
// ===== library types =====

// folder: Modbus Polling Engine

TYPE "typeMasterData"
VERSION : 0.1
   STRUCT
      Done : Bool;
      Busy : Bool;
      Error : Bool;
      locked : Bool;
      Mode : USInt;
      Status : Int;
      "Slave ID" : UInt;
      "Register Address" : UDInt;
      Length : UInt;
      RequestID : UInt;
      Data : Array[0..299] of Byte;
   END_STRUCT;
END_TYPE

// folder: (top level)

FUNCTION_BLOCK "PollTosibox"   // FB1, SCL
{ S7_Optimized_Access := 'TRUE' }
VERSION : 0.1
   VAR_INPUT
      slaveId : Int;   // modbus slave id
   END_VAR
   VAR_OUTPUT
      latitude : LReal;
      longitude : LReal;
      UTCTime : LReal;
   END_VAR
   VAR_IN_OUT
      modbusInterface : "typeMasterData";
   END_VAR
   VAR
      statData : Array[0..11] of Int;
      statLat : Array[0..7] of Byte;
      statLon : Array[0..7] of Byte;
      statUTC : Array[0..7] of Byte;
   END_VAR
   VAR_TEMP
      tempStatus : Int;
      tempPos : DInt;
   END_VAR
BEGIN
   //=============================================================================
   // AWC Inc.
   // (c)Copyright 2015 All Rights Reserved
   //-----------------------------------------------------------------------------
   // Library: (that the source is dedicated to)
   // Tested with: 1500 Family, 1200 Family
   // Engineering: TIA Portal v13 SP1 upd7
   // Restrictions: None
   // Requirements: s7 1200 or 1500 family depending on number used
   // Functionality: Get Modbus Values from TosiMox
   // 
   // 
   // 
   // 
   //-----------------------------------------------------------------------------
   // Change log table:
   // 01.00.00 07/30/2020 Created by Matt Paulissen
   //=============================================================================
   //
   "LargeModbusPoll"(slaveId:=1,
                     address:=40001,
                     data=>#statData,
                     status=>#tempStatus,
                     modbusInterface:=#modbusInterface);
   //Parse Latitude
   #statLat[0] := #statData[3].%B1;
   #statLat[1] := #statData[3].%B0;
   #statLat[2] := #statData[2].%B1;
   #statLat[3] := #statData[2].%B0;
   #statLat[4] := #statData[1].%B1;
   #statLat[5] := #statData[1].%B0;
   #statLat[6] := #statData[0].%B1;
   #statLat[7] := #statData[0].%B0;

   #tempPos := 0;
   #tempStatus := Deserialize(SRC_ARRAY := #statLat, DEST_VARIABLE => #latitude, POS := #tempPos);
   //Parse Longitude
   #statLon[0] := #statData[7].%B1;
   #statLon[1] := #statData[7].%B0;
   #statLon[2] := #statData[6].%B1;
   #statLon[3] := #statData[6].%B0;
   #statLon[4] := #statData[5].%B1;
   #statLon[5] := #statData[5].%B0;
   #statLon[6] := #statData[4].%B1;
   #statLon[7] := #statData[4].%B0;

   #tempPos := 0;
   #tempStatus := Deserialize(SRC_ARRAY := #statLon, DEST_VARIABLE => #longitude, POS := #tempPos);

   //Parse Time
   #statUTC[0] := #statData[11].%B1;
   #statUTC[1] := #statData[11].%B0;
   #statUTC[2] := #statData[10].%B1;
   #statUTC[3] := #statData[10].%B0;
   #statUTC[4] := #statData[9].%B1;
   #statUTC[5] := #statData[9].%B0;
   #statUTC[6] := #statData[8].%B1;
   #statUTC[7] := #statData[8].%B0;

   #tempPos := 0;
   #tempStatus := Deserialize(SRC_ARRAY := #statUTC, DEST_VARIABLE => #UTCTime, POS := #tempPos);
END_FUNCTION_BLOCK

FUNCTION "LargeModbusPoll" : Void   // FC892, SCL
{ S7_Optimized_Access := 'TRUE' }
VERSION : 0.1
   VAR_INPUT
      slaveId : Int;   // modbus slave id
      address : UInt;   // starting modbus register address
   END_VAR
   VAR_OUTPUT
      data : Variant;   // <uint><int><word><dword><real>
      status : Int;   // status of modbus read
   END_VAR
   VAR_IN_OUT
      modbusInterface : "typeMasterData";
   END_VAR
   VAR_TEMP
      tempPosition : DInt;
      tempStatus : Int;
      tempMode : USInt;
      tempAddress : UInt;
   END_VAR
BEGIN
   //=============================================================================
   // AWC Inc.
   // (c)Copyright 2018 All Rights Reserved
   //-----------------------------------------------------------------------------
   // Library: (that the source is dedicated to)
   // Tested with: 1500 Family, 1200 Family
   // Engineering: TIA Portal v13 SP1 upd7
   // Restrictions: None
   // Requirements: s7 1200 or 1500 family depending on number used
   // Functionality: Get Modbus Input Variant UDT
   // 
   // 
   // 
   // 
   //-----------------------------------------------------------------------------
   // Change log table:
   // 01.00.00 05/17/2018 Created by Matt Paulissen
   // 01.00.02 09/21/2018 Added request ID to detect stuck lock
   // 01.01.06 09/29/2020 Added extended modbus addressing
   //=============================================================================

   //Check for lock
   IF (NOT #modbusInterface.locked) THEN
       //Move Register and Slave address to Modbus Register
       #modbusInterface."Slave ID" := #slaveId;
       #modbusInterface."Register Address" := #address;

       //Get UDT length in bytes
       #tempStatus := Serialize(SRC_VARIABLE := #data, DEST_ARRAY => #modbusInterface.Data, POS := #tempPosition);
       IF (#tempStatus <> 0) THEN  //Exit instruction if UDT cannot be processed by the modbus interface
           RETURN;
       END_IF;
       //Get number of registers needed to poll entire UDT
       CASE #address OF
           1..9999, 10001..19999:  //Edge case for boolean values
               #tempPosition := #tempPosition * 8; //Multiply bytes by 8 to get bits
           50000..59999:  //Edge case for extended addressing
               #modbusInterface.Mode := 104;
               #modbusInterface."Register Address" := #address - 40001;
               IF ((#tempPosition MOD 2) = 0) THEN
                   #tempPosition := #tempPosition / 2;
               ELSE
                   #tempPosition := (#tempPosition / 2) + 1;
               END_IF;
           ELSE  //Normal registers
               #modbusInterface.Mode := 0;
               IF ((#tempPosition MOD 2) = 0) THEN
                   #tempPosition := #tempPosition / 2;
               ELSE
                   #tempPosition := (#tempPosition / 2) + 1;
               END_IF;
       END_CASE;
       #modbusInterface.Length := #tempPosition;
       #modbusInterface.locked := TRUE;
       #modbusInterface.RequestID += 1;
       RETURN;
   END_IF;
   //Edge case handling for extended modbus addressing
   IF (#address >= 50000 AND #address <= 59999) THEN
       #tempAddress := #address - 40001;
       #tempMode := 104;
   ELSE
       #tempAddress := #address;
       #tempMode := 0;
   END_IF;
   IF ((#modbusInterface.locked)
       AND (
       (#modbusInterface."Slave ID" = #slaveId)
       AND (#modbusInterface."Register Address" = #tempAddress)
       AND (#modbusInterface.Mode = #tempMode))
       )
   THEN
       IF (#modbusInterface.Done) THEN
           //Deserialize to output
           #tempStatus := Deserialize(SRC_ARRAY := #modbusInterface.Data, DEST_VARIABLE => #data, POS := #tempPosition);
           #modbusInterface.locked := FALSE;
           #status := #modbusInterface.Status;
       END_IF;
       IF (#modbusInterface.Error) THEN
           //TODO: error handling for variant????
           #modbusInterface.locked := 0;
           #status := #modbusInterface.Status;
       END_IF;
   END_IF;
END_FUNCTION

FUNCTION "GeneralModbusWrite" : Void   // FC893, SCL
{ S7_Optimized_Access := 'TRUE' }
VERSION : 0.1
   VAR_INPUT
      slaveId : Int;   // modbus slave id
      address : UInt;   // starting modbus register address
      write : Bool;   // write data to register
      data : Variant;   // value to write to modbus register
      swappedFloatingPoint : Bool;   // set to true for word swapped floating point
   END_VAR
   VAR_OUTPUT
      status : Word;
   END_VAR
   VAR_IN_OUT
      modbusInterface : "typeMasterData";
   END_VAR
   VAR_TEMP
      tempdWord : DWord;
      tempUint : UInt;
      tempInt : Int;
      tempWord : Word;
      tempReal : Real;
      tempBool : Bool;
      tempStatus : Int;
      tempPos : DInt;
   END_VAR
   VAR CONSTANT
      WRITE_OK : Word := 16#7000;
   END_VAR
BEGIN
   //=============================================================================
   // AWC Inc.
   // (c)Copyright 2015 All Rights Reserved
   //-----------------------------------------------------------------------------
   // Library: (that the source is dedicated to)
   // Tested with: 1500 Family, 1200 Family
   // Engineering: TIA Portal v13 SP1 upd7
   // Restrictions: None
   // Requirements: s7 1200 or 1500 family depending on number used
   // Functionality: Get Modbus Input
   // 
   // 
   // 
   // 
   //-----------------------------------------------------------------------------
   // Change log table:
   // 01.00.00 08/09/2017 Created by Matt Paulissen
   // 01.00.01 08/23/2017 Added ability to set failover value
   // 01.00.02 09/21/2018 Added request ID to detect stuck lock
   // 01.01.01 01/25/2019 Added ability to write to coils
   // 01.01.07 03/16/2021 Bug Fix for writing single coil
   //=============================================================================

   //Check for lock
   IF ((NOT #modbusInterface.locked) AND (#write)) THEN
       //Move Register and Slave address to Modbus Register
       #modbusInterface."Slave ID" := #slaveId;
       #modbusInterface."Register Address" := #address;
       #modbusInterface.Mode := 1;
       CASE TypeOf(#data) OF
           UInt:
               #modbusInterface.Length := 1;
               //VariantGet(SRC:=#data,
               //           DST=>#tempUint);
               #tempStatus := Serialize(SRC_VARIABLE := #data, DEST_ARRAY => #modbusInterface.Data, POS := #tempPos);

               //#modbusInterface.Data[0] := #tempUint;
           Int:
               #modbusInterface.Length := 1;
               // VariantGet(SRC := #data,
               //            DST => #tempInt);
               // #modbusInterface.Data[0] := INT_TO_UINT(IN:=#tempInt);
               #tempStatus := Serialize(SRC_VARIABLE := #data, DEST_ARRAY => #modbusInterface.Data, POS := #tempPos);
           Word:
               #modbusInterface.Length := 1;
               // VariantGet(SRC := #data,
               //            DST => #tempWord);
               // #modbusInterface.Data[0] := WORD_TO_UINT(IN := #tempWord);
               #tempStatus := Serialize(SRC_VARIABLE := #data, DEST_ARRAY => #modbusInterface.Data, POS := #tempPos);
           DWord:
               #modbusInterface.Length := 2;
               VariantGet(SRC := #data,
                          DST => #tempdWord);
               IF #swappedFloatingPoint THEN
                   // Swapped 
                   #modbusInterface.Data[2] := #tempdWord.%B3;
                   #modbusInterface.Data[3] := #tempdWord.%B2;
                   #modbusInterface.Data[0] := #tempdWord.%B1;
                   #modbusInterface.Data[1] := #tempdWord.%B0;
               ELSE
                   //Consecutive
                   #modbusInterface.Data[3] := #tempdWord.%B0;
                   #modbusInterface.Data[2] := #tempdWord.%B1;
                   #modbusInterface.Data[1] := #tempdWord.%B2;
                   #modbusInterface.Data[0] := #tempdWord.%B3;
               END_IF;
           Real:
               #modbusInterface.Length := 2;
               VariantGet(SRC := #data,
                          DST => #tempReal);
               #tempdWord := REAL_TO_DWORD(IN:=#tempReal);
               IF #swappedFloatingPoint THEN
                   // Swapped 
                   #modbusInterface.Data[2] := #tempdWord.%B3;
                   #modbusInterface.Data[3] := #tempdWord.%B2;
                   #modbusInterface.Data[0] := #tempdWord.%B1;
                   #modbusInterface.Data[1] := #tempdWord.%B0;
               ELSE
                   //Consecutive
                   #modbusInterface.Data[3] := #tempdWord.%B0;
                   #modbusInterface.Data[2] := #tempdWord.%B1;
                   #modbusInterface.Data[1] := #tempdWord.%B2;
                   #modbusInterface.Data[0] := #tempdWord.%B3;
               END_IF;
           Bool:
               #modbusInterface.Length := 1;
               VariantGet(SRC := #data,
                          DST => #tempBool);
               // Cleared buffer to fix bug during single coil writes
               #modbusInterface.Data[0] := 0;
               #modbusInterface.Data[1] := 0;
               #modbusInterface.Data[0].%X0 := #tempBool;
           ELSE  // Statement section ELSE
               ;
       END_CASE;
       #modbusInterface.locked := TRUE;
       #modbusInterface.RequestID += 1;
       RETURN;
   END_IF;
   IF ((#modbusInterface.locked)
       AND (
       (#modbusInterface."Slave ID" = #slaveId)
       AND (#modbusInterface."Register Address" = #address)
       AND (#modbusInterface.Mode = 1))
       )
   THEN
       IF (#modbusInterface.Done) THEN
           //Inspect type of output and set correct type of input in modbus register
           #status := #WRITE_OK;
           #modbusInterface.locked := FALSE;
       END_IF;
       IF (#modbusInterface.Error) THEN
           #status := #modbusInterface.Status;
           #modbusInterface.locked := false;
       END_IF;
   END_IF;
END_FUNCTION

FUNCTION "Mag6/8000" : Void   // FC896, SCL
{ S7_Optimized_Access := 'TRUE' }
VERSION : 0.1
   VAR_INPUT
      slaveId : Int;   // modbus slave id
   END_VAR
   VAR_OUTPUT
      velocity : Variant;   // current velocity <real>
      flow : Variant;   // current flow <real>
      totalizer : Variant;   // totalizer <array[0..2] of UDINT>
   END_VAR
   VAR_IN_OUT
      modbusInterface : "typeMasterData";
   END_VAR
   VAR_TEMP
      tempStatus : Int;
   END_VAR
BEGIN
   //=============================================================================
   // AWC Inc.
   // (c)Copyright 2015 All Rights Reserved
   //-----------------------------------------------------------------------------
   // Library: (that the source is dedicated to)
   // Tested with: 1500 Family, 1200 Family
   // Engineering: TIA Portal v13 SP1 upd7
   // Restrictions: None
   // Requirements: s7 1200 or 1500 family depending on number used
   // Functionality: Get Modbus Values from Siemens Mag6000 or 8000
   // 
   // 
   // 
   // 
   //-----------------------------------------------------------------------------
   // Change log table:
   // 01.00.00 01/14/2019 Created by Matt Paulissen
   //=============================================================================
   //Current Velocity
   "GeneralModbusPoll"(slaveId:=#slaveId,
                       address:=42999,
                       swappedFloatingPoint:=false,
                       substituteValue:=0.0,
                       data=>#velocity,
                       modbusInterface:=#modbusInterface);
   //Current Flow
   "GeneralModbusPoll"(slaveId := #slaveId,
                       address := 43001,
                       swappedFloatingPoint := false,
                       substituteValue := 0.0,
                       data => #flow,
                       modbusInterface := #modbusInterface);
   //Totalizer
   "LargeModbusPoll"(slaveId:=#slaveId,
                     address:=43016
                     ,
                     data=>#totalizer,
                     status=> #tempStatus,
                     modbusInterface:=#modbusInterface);
END_FUNCTION

// folder: Cameron

FUNCTION "NuFlo" : Void   // FC897, SCL
{ S7_Optimized_Access := 'TRUE' }
VERSION : 0.1
   VAR_INPUT
      slaveId : Int;   // modbus slave id
   END_VAR
   VAR_OUTPUT
      currentFlow : Variant;   // current flow <real>
      currentTotal : Variant;   // current total <real>
      grandTotal : Variant;   // grand total <real>
   END_VAR
   VAR_IN_OUT
      modbusInterface : "typeMasterData";
   END_VAR
BEGIN
   //=============================================================================
   // AWC Inc.
   // (c)Copyright 2015 All Rights Reserved
   //-----------------------------------------------------------------------------
   // Library: (that the source is dedicated to)
   // Tested with: 1500 Family, 1200 Family
   // Engineering: TIA Portal v13 SP1 upd7
   // Restrictions: None
   // Requirements: s7 1200 or 1500 family depending on number used
   // Functionality: Get Modbus Values from Cameron Nu Flo
   // 
   // 
   // 
   // 
   //-----------------------------------------------------------------------------
   // Change log table:
   // 01.00.00 01/08/2019 Created by Matt Paulissen
   //=============================================================================
   //Current Flow
   "GeneralModbusPoll"(slaveId:=#slaveId,
                       address:=48013,
                       swappedFloatingPoint:=false,
                       substituteValue:=0.0,
                       data=>#currentFlow,
                       modbusInterface:=#modbusInterface);
   //Current Total
   "GeneralModbusPoll"(slaveId := #slaveId,
                       address := 48027,
                       swappedFloatingPoint := false,
                       substituteValue := 0.0,
                       data => #currentTotal,
                       modbusInterface := #modbusInterface);
   //Grand Total
   "GeneralModbusPoll"(slaveId := #slaveId,
                       address := 48011,
                       swappedFloatingPoint := false,
                       substituteValue := 0.0,
                       data => #grandTotal,
                       modbusInterface := #modbusInterface);
END_FUNCTION

// folder: ElectroLab

FUNCTION "LevelStick2100" : Void   // FC898, SCL
{ S7_Optimized_Access := 'TRUE' }
VERSION : 0.1
   VAR_INPUT
      slaveId : Int;   // modbus slave id
   END_VAR
   VAR_OUTPUT
      level : Variant;   // current level <uint>
      interfaceLevel : Variant;   // current interface level <uint>
   END_VAR
   VAR_IN_OUT
      modbusInterface : "typeMasterData";
   END_VAR
BEGIN
   //=============================================================================
   // AWC Inc.
   // (c)Copyright 2015 All Rights Reserved
   //-----------------------------------------------------------------------------
   // Library: (that the source is dedicated to)
   // Tested with: 1500 Family, 1200 Family
   // Engineering: TIA Portal v13 SP1 upd7
   // Restrictions: None
   // Requirements: s7 1200 or 1500 family depending on number used
   // Functionality: Get Modbus Values from Electrolab 2100
   // 
   // 
   // 
   // 
   //-----------------------------------------------------------------------------
   // Change log table:
   // 01.00.00 01/14/2019 Created by Matt Paulissen
   //=============================================================================
   //Current Velocity
   "GeneralModbusPoll"(slaveId:=#slaveId,
                       address:=43991,
                       swappedFloatingPoint:=false,
                       substituteValue:=0.0,
                       data=>#level,
                       modbusInterface:=#modbusInterface);
   "GeneralModbusPoll"(slaveId := #slaveId,
                       address := 43992,
                       swappedFloatingPoint := false,
                       substituteValue := 0.0,
                       data => #interfaceLevel,
                       modbusInterface := #modbusInterface);
END_FUNCTION

// folder: Modbus Polling Engine

FUNCTION_BLOCK "ModbusRtuEngine"   // FB6, LAD
{ S7_Optimized_Access := 'TRUE' }
VERSION : 0.1
// S7 1200 version of modbus polling engine.  Changed the Modbus Master to an MB_Master
   VAR_INPUT
      port : Port;
      baudRate : UDInt;
      parity : UInt;
      FirstScan : Bool;
      Reset : Bool;
   END_VAR
   VAR_OUTPUT
      Status : Int;
   END_VAR
   VAR_IN_OUT
      masterInterface : "typeMasterData";
   END_VAR
   VAR
      statPrevious : Int;
      statCurrent : Int;
      statIndex : Int;
      statRequestID : UInt;
      Comm_Load_Status : Int;
      Comm_Load_Done : Bool;
      Comm_Load_Error : Bool;
      instStuckInterfaceTimer : TON_TIME;
      instReinitilizeTimer : TON_TIME;
      instCommLoad : Modbus_Comm_Load;
      instMaster : Modbus_Master;
      inst7002Timeout : TON_TIME;
   END_VAR
   VAR_TEMP
      tempServerStatus : Int;
   END_VAR
   VAR CONSTANT
      UNITIALIZED : Int := 0;
      INITIALIZING_PORT : Int := 1;
      POLLING : Int := 2;
      POLLING_DONE : Int := 3;
   END_VAR
   VAR_TEMP   // added for the SCL form of the ladder/FBD networks
      _w1 : Bool;
   END_VAR
BEGIN

REGION Network 1: Run Comm Load
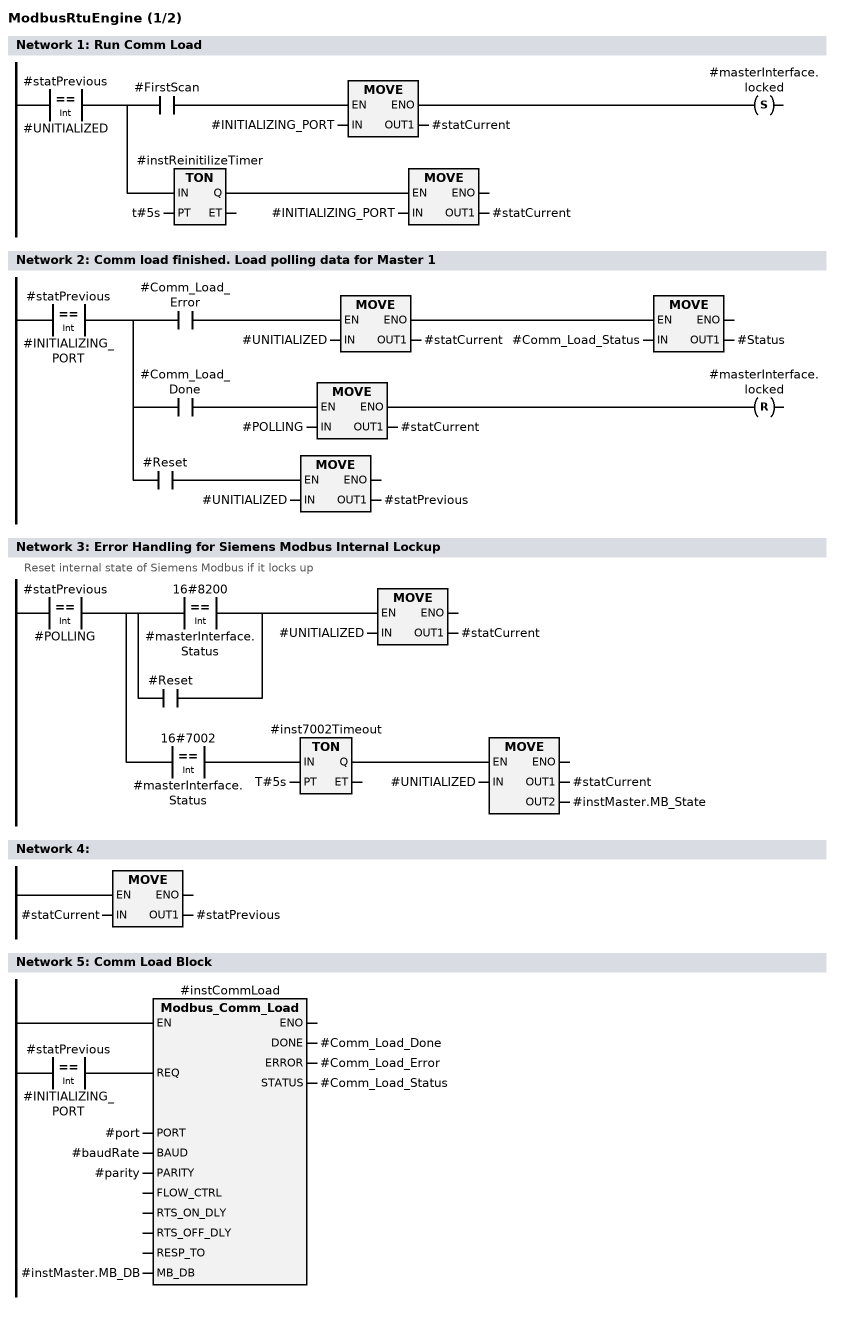
   #_w1 := #statPrevious = #UNITIALIZED;
   IF #_w1 AND #FirstScan THEN
       #statCurrent := #INITIALIZING_PORT;
       #masterInterface.locked := TRUE;
   END_IF;
   #instReinitilizeTimer(IN := #_w1, PT := t#5s);   // TON
   IF #instReinitilizeTimer.Q THEN #statCurrent := #INITIALIZING_PORT; END_IF;
END_REGION

REGION Network 2: Comm load finished. Load polling data for Master 1
   RUNG wire#powerrail
      { S7_Templates := "SrcType := Int" } EQ_Contact(in1 := #statPrevious, in2 := #INITIALIZING_PORT)
      wire#w1
      Contact( #Comm_Load_Error )
      Move(in := #UNITIALIZED, out1 => #statCurrent)
      Move(in := #Comm_Load_Status, out1 => #Status)
   END_RUNG
   RUNG wire#w1
      Contact( #Comm_Load_Done )
      Move(in := #POLLING, out1 => #statCurrent)
      R_Coil( #masterInterface.locked )
   END_RUNG
   RUNG wire#w1
      Contact( #Reset )
      Move(in := #UNITIALIZED, out1 => #statPrevious)
   END_RUNG
   // the same network as SCL:
   #_w1 := #statPrevious = #INITIALIZING_PORT;
   IF #_w1 AND #Comm_Load_Error THEN
       #statCurrent := #UNITIALIZED;
       #Status := #Comm_Load_Status;
   END_IF;
   IF #_w1 AND #Comm_Load_Done THEN
       #statCurrent := #POLLING;
       #masterInterface.locked := FALSE;
   END_IF;
   IF #_w1 AND #Reset THEN #statPrevious := #UNITIALIZED; END_IF;
END_REGION

REGION Network 3: Error Handling for Siemens Modbus Internal Lockup
   // Reset internal state of Siemens Modbus if it locks up
   #_w1 := #statPrevious = #POLLING;
   IF #_w1 AND ((16#8200 = #masterInterface.Status) OR #Reset) THEN #statCurrent := #UNITIALIZED; END_IF;
   #inst7002Timeout(IN := #_w1 AND (16#7002 = #masterInterface.Status), PT := T#5s);   // TON
   IF #inst7002Timeout.Q THEN
       #statCurrent := #UNITIALIZED;
       #instMaster.MB_State := #UNITIALIZED;
   END_IF;
END_REGION

REGION Network 4
   RUNG wire#powerrail
      Move(in := #statCurrent, out1 => #statPrevious)
   END_RUNG
   // the same network as SCL:
   #statPrevious := #statCurrent;
END_REGION

REGION Network 5: Comm Load Block
   #instCommLoad(REQ := #statPrevious = #INITIALIZING_PORT,   // Modbus_Comm_Load
                 PORT := #port,
                 BAUD := #baudRate,
                 PARITY := #parity,
                 MB_DB := #instMaster.MB_DB,
                 DONE => #Comm_Load_Done,
                 ERROR => #Comm_Load_Error,
                 STATUS => #Comm_Load_Status);
END_REGION

REGION Network 6: Master Instance 1
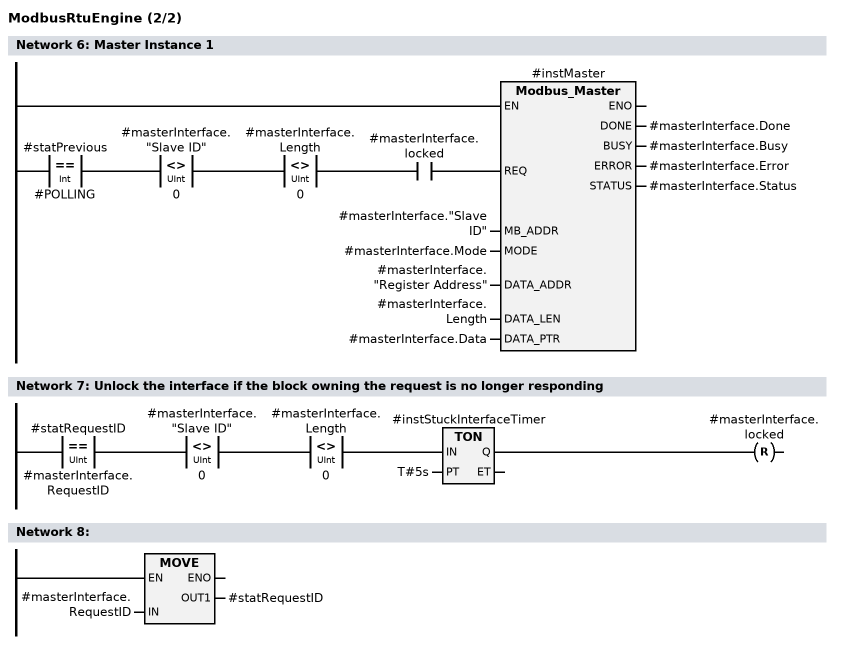
   #instMaster(REQ := (#statPrevious = #POLLING) AND (#masterInterface."Slave ID" <> 0) AND (#masterInterface.Length <> 0) AND #masterInterface.locked,   // Modbus_Master
               MB_ADDR := #masterInterface."Slave ID",
               MODE := #masterInterface.Mode,
               DATA_ADDR := #masterInterface."Register Address",
               DATA_LEN := #masterInterface.Length,
               DATA_PTR := #masterInterface.Data,
               DONE => #masterInterface.Done,
               BUSY => #masterInterface.Busy,
               ERROR => #masterInterface.Error,
               STATUS => #masterInterface.Status);
END_REGION

REGION Network 7: Unlock the interface if the block owning the request is no longer responding
   #instStuckInterfaceTimer(IN := (#statRequestID = #masterInterface.RequestID) AND (#masterInterface."Slave ID" <> 0) AND (#masterInterface.Length <> 0),   // TON
                           PT := T#5s);
   IF #instStuckInterfaceTimer.Q THEN #masterInterface.locked := FALSE; END_IF;
END_REGION

REGION Network 8
   RUNG wire#powerrail
      Move(in := #masterInterface.RequestID, out1 => #statRequestID)
   END_RUNG
   // the same network as SCL:
   #statRequestID := #masterInterface.RequestID;
END_REGION
END_FUNCTION_BLOCK

FUNCTION_BLOCK "ModbusTCPEngine"   // FB22, LAD
{ S7_Optimized_Access := 'TRUE' }
VERSION : 0.1
   VAR_INPUT
      port : Hw_Any;   // hardware identifier of port
      connectionId : Conn_Ouc;
      tcpPort : UInt;
      ipOne : Byte;   // ip octet one
      ipTwo : Byte;   // ip octet two
      ipThree : Byte;   // ip octet three
      ipFour : Byte;   // ip octet four
   END_VAR
   VAR_OUTPUT
      Status : Int;
   END_VAR
   VAR_IN_OUT
      masterInterface : "typeMasterData";
   END_VAR
   VAR
      instClient : MB_CLIENT;
      connection : TCON_IP_v4;
      statRequestID : UInt;
      instStuckInterfaceTimer : TON_TIME;
   END_VAR
   VAR CONSTANT
      UNITIALIZED : Int := 0;
      INITIALIZING_PORT : Int := 1;
      POLLING_ONE : Int := 2;
      POLLING_DONE_ONE : Int := 3;
      POLLING_TWO : Int := 4;
      POLLING_TWO_DONE : Int := 5;
   END_VAR
   // connection.ConnectionType := 11;
   // connection.ActiveEstablished := 1;
   // connection.RemotePort := 502;
   // connection.LocalPort := 502;
BEGIN

REGION Network 1: Move ip address from interface to static tcon_ip_v4
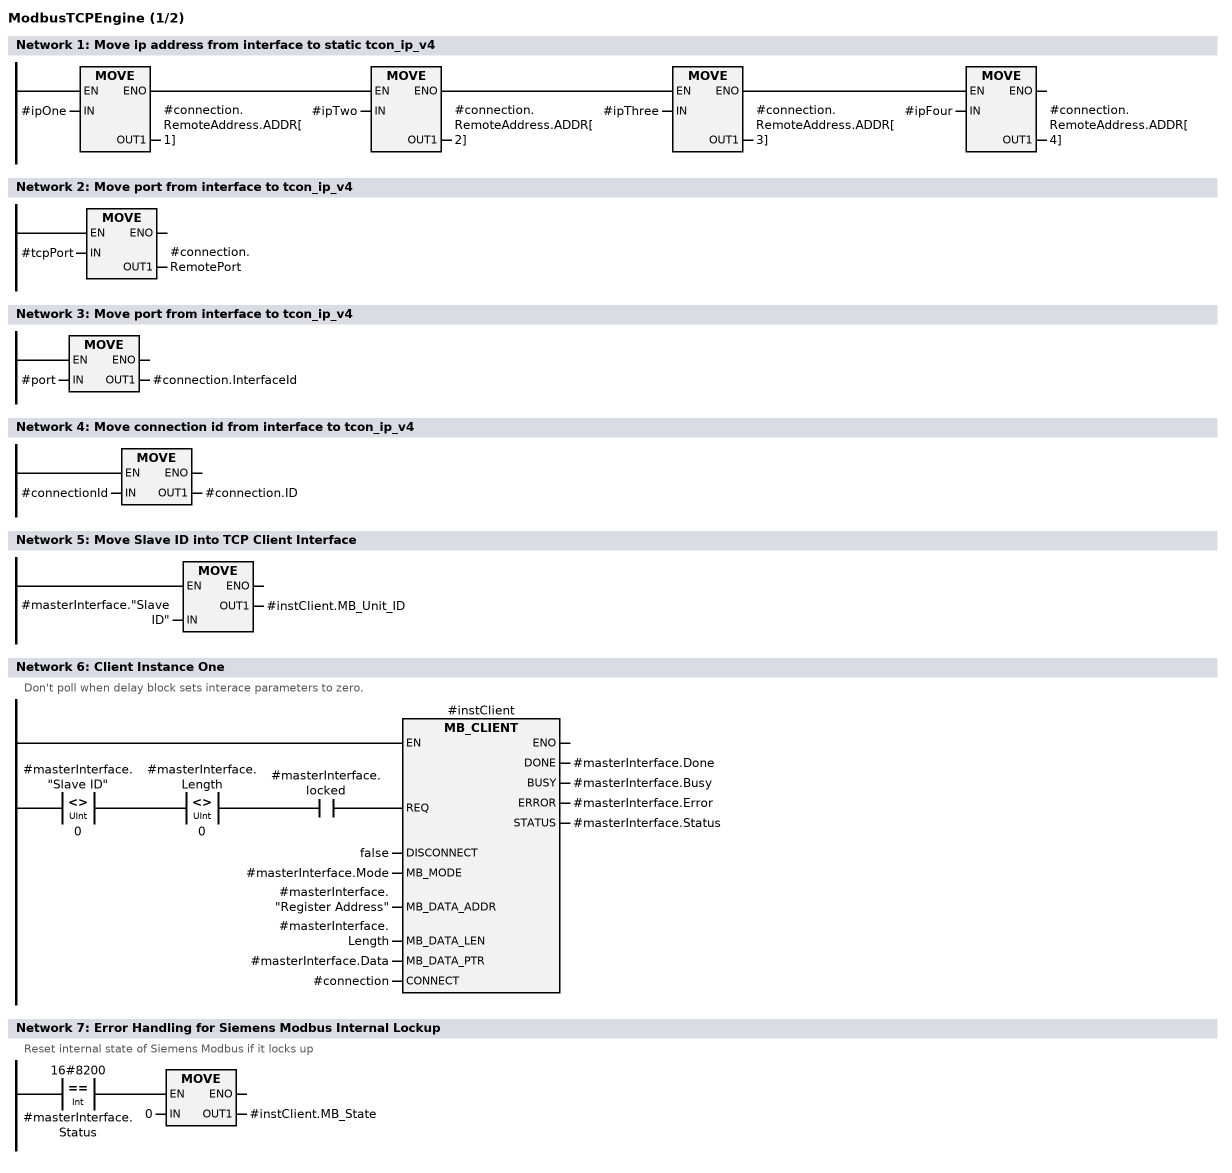
   RUNG wire#powerrail
      Move(in := #ipOne, out1 => #connection.RemoteAddress.ADDR[1])
      Move(in := #ipTwo, out1 => #connection.RemoteAddress.ADDR[2])
      Move(in := #ipThree, out1 => #connection.RemoteAddress.ADDR[3])
      Move(in := #ipFour, out1 => #connection.RemoteAddress.ADDR[4])
   END_RUNG
   // the same network as SCL:
   #connection.RemoteAddress.ADDR[1] := #ipOne;
   #connection.RemoteAddress.ADDR[2] := #ipTwo;
   #connection.RemoteAddress.ADDR[3] := #ipThree;
   #connection.RemoteAddress.ADDR[4] := #ipFour;
END_REGION

REGION Network 2: Move port from interface to tcon_ip_v4
   RUNG wire#powerrail
      Move(in := #tcpPort, out1 => #connection.RemotePort)
   END_RUNG
   // the same network as SCL:
   #connection.RemotePort := #tcpPort;
END_REGION

REGION Network 3: Move port from interface to tcon_ip_v4
   RUNG wire#powerrail
      Move(in := #port, out1 => #connection.InterfaceId)
   END_RUNG
   // the same network as SCL:
   #connection.InterfaceId := #port;
END_REGION

REGION Network 4: Move connection id from interface to tcon_ip_v4
   RUNG wire#powerrail
      Move(in := #connectionId, out1 => #connection.ID)
   END_RUNG
   // the same network as SCL:
   #connection.ID := #connectionId;
END_REGION

REGION Network 5: Move Slave ID into TCP Client Interface
   RUNG wire#powerrail
      Move(in := #masterInterface."Slave ID", out1 => #instClient.MB_Unit_ID)
   END_RUNG
   // the same network as SCL:
   #instClient.MB_Unit_ID := #masterInterface."Slave ID";
END_REGION

REGION Network 6: Client Instance One
   // Don't poll when delay block sets interace parameters to zero.
   #instClient(REQ := (#masterInterface."Slave ID" <> 0) AND (#masterInterface.Length <> 0) AND #masterInterface.locked,   // MB_CLIENT
               DISCONNECT := false,
               MB_MODE := #masterInterface.Mode,
               MB_DATA_ADDR := #masterInterface."Register Address",
               MB_DATA_LEN := #masterInterface.Length,
               MB_DATA_PTR := #masterInterface.Data,
               CONNECT := #connection,
               DONE => #masterInterface.Done,
               BUSY => #masterInterface.Busy,
               ERROR => #masterInterface.Error,
               STATUS => #masterInterface.Status);
END_REGION

REGION Network 7: Error Handling for Siemens Modbus Internal Lockup
   // Reset internal state of Siemens Modbus if it locks up
   RUNG wire#powerrail
      { S7_Templates := "SrcType := Int" } EQ_Contact(in1 := 16#8200, in2 := #masterInterface.Status)
      Move(in := 0, out1 => #instClient.MB_State)
   END_RUNG
   // the same network as SCL:
   IF 16#8200 = #masterInterface.Status THEN #instClient.MB_State := 0; END_IF;
END_REGION

REGION Network 8: Unlock the interface if the block owning the request is no longer responding
   // Modbus Polling Delay block sets interfaces to zero.  Don't want to unlock interface if this block is holding it.
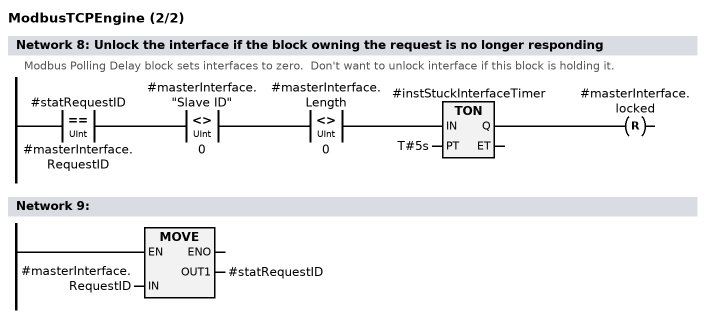
   #instStuckInterfaceTimer(IN := (#statRequestID = #masterInterface.RequestID) AND (#masterInterface."Slave ID" <> 0) AND (#masterInterface.Length <> 0),   // TON
                           PT := T#5s);
   IF #instStuckInterfaceTimer.Q THEN #masterInterface.locked := FALSE; END_IF;
END_REGION

REGION Network 9
   RUNG wire#powerrail
      Move(in := #masterInterface.RequestID, out1 => #statRequestID)
   END_RUNG
   // the same network as SCL:
   #statRequestID := #masterInterface.RequestID;
END_REGION
END_FUNCTION_BLOCK

// folder: Modbus Polling Engine/Modbus Polling Functions

FUNCTION "GeneralModbusPoll" : Void   // FC11, SCL
{ S7_Optimized_Access := 'TRUE' }
VERSION : 0.1
   VAR_INPUT
      slaveId : Int;   // modbus slave id
      address : UInt;   // starting modbus register address
      swappedFloatingPoint : Bool;   // set to true for word swapped floating point
      substituteValue : Real;   // value returned on polling error
   END_VAR
   VAR_OUTPUT
      data : Variant;   // <uint><int><word><dword><real><bool>
   END_VAR
   VAR_IN_OUT
      modbusInterface : "typeMasterData";
   END_VAR
   VAR_TEMP
      tempArray : Array[0..3] of Byte;
      tempDWord : DWord;
      tempStatus : Int;
      tempPos : DInt;
      tempBool : Bool;
   END_VAR
BEGIN
   //=============================================================================
   // AWC Inc.
   // (c)Copyright 2015 All Rights Reserved
   //-----------------------------------------------------------------------------
   // Library: (that the source is dedicated to)
   // Tested with: 1500 Family, 1200 Family
   // Engineering: TIA Portal v13 SP1 upd7
   // Restrictions: None
   // Requirements: s7 1200 or 1500 family depending on number used
   // Functionality: Get Modbus Input
   // 
   // 
   // 
   // 
   //-----------------------------------------------------------------------------
   // Change log table:
   // 01.00.00 08/09/2017 Created by Matt Paulissen
   // 01.00.01 08/23/2017 Added ability to set failover value
   // 01.00.02 09/21/2018 Added request ID to detect stuck lock
   // 01.01.01 01/25/2019 Added ability to read contacts
   //=============================================================================

   //Check for lock
   IF (NOT #modbusInterface.locked) THEN
       //Move Register and Slave address to Modbus Register
       #modbusInterface."Slave ID" := #slaveId;
       #modbusInterface."Register Address" := #address;
       #modbusInterface.Mode := 0;
       CASE TypeOf(#data) OF
           UInt:
               #modbusInterface.Length := 1;
           Int:
               #modbusInterface.Length := 1;
           Word:
               #modbusInterface.Length := 1;
           DWord:
               #modbusInterface.Length := 2;
           Real:
               #modbusInterface.Length := 2;
           Bool:
               #modbusInterface.Length := 1;
           ELSE  // Statement section ELSE
               ;
       END_CASE;
       #modbusInterface.locked := TRUE;
       #modbusInterface.RequestID += 1;
       RETURN;
   END_IF;
   IF ((#modbusInterface.locked)
       AND (
       (#modbusInterface."Slave ID" = #slaveId)
       AND (#modbusInterface."Register Address" = #address)
       AND (#modbusInterface.Mode = 0))
       )
   THEN
       IF (#modbusInterface.Done) THEN
           //Inspect type of output and set correct type of input in modbus register
           CASE TypeOf(#data) OF
               UInt:
                   #tempStatus := Deserialize(SRC_ARRAY := #modbusInterface.Data,
                                              DEST_VARIABLE => #data,
                                              POS := #tempPos);
               Int:
                   #tempStatus := Deserialize(SRC_ARRAY := #modbusInterface.Data,
                                              DEST_VARIABLE => #data,
                                              POS := #tempPos);
               Word:
                   #tempStatus := Deserialize(SRC_ARRAY := #modbusInterface.Data,
                                              DEST_VARIABLE => #data,
                                              POS := #tempPos);
               DWord:
                   IF #swappedFloatingPoint THEN
                       // Swapped 
                       #tempArray[3] := #modbusInterface.Data[1];
                       #tempArray[2] := #modbusInterface.Data[0];
                       #tempArray[1] := #modbusInterface.Data[3];
                       #tempArray[0] := #modbusInterface.Data[2];
                       #tempStatus := Deserialize(SRC_ARRAY := #tempArray,
                                                  DEST_VARIABLE => #data,
                                                  POS := #tempPos);
                   ELSE
                       //Consecutive
                       #tempStatus := Deserialize(SRC_ARRAY := #modbusInterface.Data,
                                                  DEST_VARIABLE => #data,
                                                  POS := #tempPos);
                   END_IF;

               Real:
                   IF #swappedFloatingPoint THEN
                       // Swapped 
                       #tempArray[3] := #modbusInterface.Data[1];
                       #tempArray[2] := #modbusInterface.Data[0];
                       #tempArray[1] := #modbusInterface.Data[3];
                       #tempArray[0] := #modbusInterface.Data[2];
                       #tempStatus := Deserialize(SRC_ARRAY := #tempArray,
                                                  DEST_VARIABLE => #data,
                                                  POS := #tempPos);

                   ELSE
                       //Consecutive
                       #tempStatus := Deserialize(SRC_ARRAY := #modbusInterface.Data,
                                                  DEST_VARIABLE => #data,
                                                  POS := #tempPos);
                   END_IF;

               Bool:
                   #tempBool := #modbusInterface.Data[0].%X0;
                   VariantPut(SRC := #tempBool,
                              DST := #data);
               ELSE  // Statement section ELSE
                   ;
           END_CASE;
           #modbusInterface.locked := FALSE;
       END_IF;
       IF (#modbusInterface.Error) THEN
           CASE TypeOf(#data) OF
               UInt:
                   VariantPut(SRC := REAL_TO_UINT(IN:=#substituteValue),
                              DST := #data);
               Int:
                   VariantPut(SRC := REAL_TO_INT(IN := #substituteValue),
                              DST := #data);
               Word:
                   VariantPut(SRC := INT_TO_WORD(IN:=TRUNC_INT(IN := #substituteValue)),
                              DST := #data);
               DWord:
                   VariantPut(SRC := REAL_TO_DWORD(IN:=#tempDWord),
                              DST := #data);
               Real:
                   VariantPut(SRC := #substituteValue,
                              DST := #data);
               Bool:
                   IF (#substituteValue <> 0.0) THEN
                       #tempBool := TRUE;
                   ELSE
                       #tempBool := FALSE;
                   END_IF;
                   VariantPut(SRC := #tempBool,
                              DST := #data);
               ELSE  // Statement section ELSE
                   ;
           END_CASE;
           #modbusInterface.locked := 0;
       END_IF;
   END_IF;
END_FUNCTION

FUNCTION "LargeModbusWrite" : Void   // FC894, SCL
{ S7_Optimized_Access := 'TRUE' }
VERSION : 0.1
   VAR_INPUT
      slaveId : Int;   // modbus slave id
      address : UInt;   // starting modbus register address
      write : Bool;   // write data to register
      data : Variant;   // value to write to modbus register
   END_VAR
   VAR_OUTPUT
      status : Word;
   END_VAR
   VAR_IN_OUT
      modbusInterface : "typeMasterData";
   END_VAR
   VAR_TEMP
      tempPosition : DInt;
      tempStatus : Int;
   END_VAR
   VAR CONSTANT
      WRITE_OK : Word := 16#7000;
   END_VAR
BEGIN
   //=============================================================================
   // AWC Inc.
   // (c)Copyright 2018 All Rights Reserved
   //-----------------------------------------------------------------------------
   // Library: (that the source is dedicated to)
   // Tested with: 1500 Family, 1200 Family
   // Engineering: TIA Portal v13 SP1 upd7
   // Restrictions: None
   // Requirements: s7 1200 or 1500 family depending on number used
   // Functionality: Write to modbus device
   // 
   // 
   // 
   // 
   //-----------------------------------------------------------------------------
   // Change log table:
   // 01.00.00 05/17/2018 Created by Matt Paulissen
   // 01.00.02 09/21/2018 Added request ID to detect stuck lock
   //=============================================================================

   //Check for lock
   IF ((NOT #modbusInterface.locked) AND (#write)) THEN
       //Move Register and Slave address to Modbus Register
       #modbusInterface."Slave ID" := #slaveId;
       #modbusInterface."Register Address" := #address;
       #modbusInterface.Mode := 1;
       //Move data to interface and get length
       #tempStatus := Serialize(SRC_VARIABLE := #data, DEST_ARRAY => #modbusInterface.Data, POS := #tempPosition);
       IF (#tempStatus <> 0) THEN  //Exit instruction if UDT cannot be processed by the modbus interface
           RETURN;
       END_IF;
       //Get number of registers needed to poll entire UDT
       CASE #address OF
           1..9999, 10001..19999:  //Edge case for boolean values
               #tempPosition := #tempPosition * 8; //Multiply bytes by 8 to get bits
           ELSE  //Normal registers
               IF ((#tempPosition MOD 2) = 0) THEN
                   #tempPosition := #tempPosition / 2;
               ELSE
                   #tempPosition := (#tempPosition / 2) + 1;
               END_IF;
       END_CASE;
       #modbusInterface.Length := #tempPosition;
       #modbusInterface.locked := TRUE;
       #modbusInterface.RequestID += 1;
       RETURN;
   END_IF;
   IF ((#modbusInterface.locked)
       AND (
       (#modbusInterface."Slave ID" = #slaveId)
       AND (#modbusInterface."Register Address" = #address)
       AND (#modbusInterface.Mode = 1))
       )
   THEN
       IF (#modbusInterface.Done) THEN
           //Inspect type of output and set correct type of input in modbus register
           #status := #WRITE_OK;
           #modbusInterface.locked := FALSE;
       END_IF;
       IF (#modbusInterface.Error) THEN
           #status := #modbusInterface.Status;
           #modbusInterface.locked := false;
       END_IF;
   END_IF;
END_FUNCTION

FUNCTION "ModbusPollingDelay" : Void   // FC895, SCL
{ S7_Optimized_Access := 'TRUE' }
VERSION : 0.1
   VAR_INPUT
      timerID : Int;   // modbus timer ID
      delayTime : Time;   // time to delay polling
   END_VAR
   VAR_IN_OUT
      modbusInterface : "typeMasterData";
   END_VAR
   VAR_TEMP
      tempPosition : DInt;
      tempStatus : Int;
      tempCurrentTime : DTL;
      tempStartTime : DTL;
      tempEndTime : DTL;
   END_VAR
BEGIN
   //=============================================================================
   // AWC Inc.
   // (c)Copyright 2018 All Rights Reserved
   //-----------------------------------------------------------------------------
   // Library: (that the source is dedicated to)
   // Tested with: 1500 Family, 1200 Family
   // Engineering: TIA Portal v13 SP1 upd7
   // Restrictions: None
   // Requirements: s7 1200 or 1500 family depending on number used
   // Functionality: Add delay to modbus polling engine
   // 
   // 
   // 
   // 
   //-----------------------------------------------------------------------------
   // Change log table:
   // 01.00.00 01/08/2019 Created by Matt Paulissen
   //=============================================================================

   //Check for lock
   IF (NOT #modbusInterface.locked) THEN
       //Create ID out of current PLC time
       #tempStatus := RD_SYS_T(#tempCurrentTime);
       //Serialize start time into interface
       #tempPosition := 0;
       #tempStatus := Serialize(SRC_VARIABLE := #tempCurrentTime, DEST_ARRAY => #modbusInterface.Data, POS := #tempPosition);
       #modbusInterface."Slave ID" := 0;
       #modbusInterface."Register Address" := #timerID;
       #modbusInterface.Mode := 0;
       #modbusInterface.Length := 0;
       #modbusInterface.locked := TRUE;
       #modbusInterface.RequestID += 1;
       RETURN;
   END_IF;
   IF ((#modbusInterface.locked)
       AND (
       (#modbusInterface."Slave ID" = 0)
       AND (#modbusInterface."Register Address" = #timerID)
       AND (#modbusInterface.Mode = 0))
       )
   THEN
       #tempPosition := 0;
       #tempStatus := Deserialize(SRC_ARRAY := #modbusInterface.Data, DEST_VARIABLE => #tempStartTime, POS := #tempPosition);
       #tempEndTime := T_ADD(IN1 := #tempStartTime, IN2 := #delayTime);
       #tempStatus := RD_SYS_T(#tempCurrentTime);
       IF (#tempCurrentTime > #tempEndTime) THEN
           #modbusInterface.locked := FALSE;
       END_IF;
   END_IF;
END_FUNCTION